// TwinCAT 3 PLC project Untitled1
// ProgramVersion: 3.1.4023.0
// libraries:
//   Tc2_Standard, * (Beckhoff Automation GmbH)
//   Tc2_System, * (Beckhoff Automation GmbH)
//   Tc2_Utilities, * (Beckhoff Automation GmbH)
//   Tc3_Module, * (Beckhoff Automation GmbH)
// project tree:
//   DUTs/ HMI_Instructions.TcDUT, IO_Struct.TcDUT, Port_Map.TcDUT (not stored), Test_Log.TcDUT
//   GVLs/ GVL_HMI.TcGVL, GVL_IO_STRUCTS.TcGVL, GVL_LOGS.TcGVL (not stored), GVL_IO.TcGVL, CONSTANTS.TcGVL
//   / PlcTask.TcTTO (not stored)
//   POUs/ FB_EXECUTE_SECTION1.TcPOU, FB_EXECUTE_SECTION2.TcPOU, INITIALIZE.TcPOU, LOG_SECTION2.TcPOU, LOG_SECTION1.TcPOU, MAIN.TcPOU, UNINITIALIZE.TcPOU, UPDATE_HMI.TcPOU, WRITE_IO_VALUES.TcPOU
// real-time tasks:
//   TASK PlcTask: cycle T#10ms, priority 20, ADS port 350
// I/O:
//   DEVICE Device 1 (EtherCAT), AmsNetId 10.14.22.198.2.1
//     C0 (EK1914) [EK1914, 2 Ch. Safety Input/Output 24V,  TwinSAFE]
//       modules: Module 1 (FSOE), Module 2 (DIO)
//       C1 (EL9410) [EL9410 E-Bus Power Supplier  (Diagnostics)]
//       C2 (EL2014) [EL2014 4Ch. Dig. Output 24V, 0,5A, Diagnostic]
//       C3 (EL1018) [EL1018 8Ch. Dig. Input 24V, 10µs]
//       C4 (EL1819) [EL1819 16Ch. Dig. Input 24V, 10µs]
//       C5 (EL1819) [EL1819 16Ch. Dig. Input 24V, 10µs]
//       C6 (EK1122-0008) [EK1122-0008 2 port EtherCAT junction M8]
//         JBC0 (EK1914) [EK1914, 2 Ch. Safety Input/Output 24V,  TwinSAFE]
//           modules: Module 1 (FSOE), Module 2 (DIO)
//           JBC1 (EL9410) [EL9410 E-Bus Power Supplier  (Diagnostics)]
//           JBC2 (EL1904) [EL1904, 4 Ch. Safety Input 24V, TwinSAFE]
//             modules: Module 1 (FSOES)
//           JBC3 (EL3174) [EL3174 4K. Ana. Eingang  +/-10V Diff., +/-20mA SingleEnded, 16 Bit]
//           JBC4 (EK1122-0008) [EK1122-0008 2 port EtherCAT junction M8]
//           JBC5 (EK1122-0008) [EK1122-0008 2 port EtherCAT junction M8]
//             JBB0 (EP3752-0000) [EP3752-0000 Acceleration Sensor]
// variable links:
//   Untitled1/Untitled1 Instance <-> Device 1 (EtherCAT)/C0 (EK1914)/C2 (EL2014)
//     PlcTask Outputs/GVL_IO.SF5_Fire_Alarm <-> DIG Outputs/Channel 2/Output
//   Untitled1/Untitled1 Instance <-> Device 1 (EtherCAT)/C0 (EK1914)/C3 (EL1018)
//     PlcTask Inputs/GVL_IO.J7_24V_Up <-> Channel 1/Input
//     PlcTask Inputs/GVL_IO.J8_24V_Up <-> Channel 3/Input
//     PlcTask Inputs/GVL_IO.J7_24V_Us <-> Channel 2/Input
//     PlcTask Inputs/GVL_IO.J8_24V_Us <-> Channel 4/Input
//   Untitled1/Untitled1 Instance <-> Device 1 (EtherCAT)/C0 (EK1914)/C4 (EL1819)
//     PlcTask Inputs/GVL_IO.J{1..6}_24V_Up <-> Channel {1..11 step 2}/Input  (6 links)
//     PlcTask Inputs/GVL_IO.J{1..6}_24V_Us <-> Channel {2..12 step 2}/Input  (6 links)
//   Untitled1/Untitled1 Instance <-> Device 1 (EtherCAT)/C0 (EK1914)/C5 (EL1819)
//     PlcTask Inputs/GVL_IO.SF1_MF_CONTINUITY <-> Channel 16/Input
//     PlcTask Inputs/GVL_IO.SF2_MF_CONTINUITY <-> Channel 15/Input
//     PlcTask Inputs/GVL_IO.SF4_Pull_Station <-> Channel 14/Input
//     PlcTask Inputs/GVL_IO.SF6_MGT_CONTINUITY <-> Channel 13/Input
//     PlcTask Inputs/GVL_IO.SF8_MGT_CONTINUITY <-> Channel 12/Input
//   Untitled1/Untitled1 Instance <-> Device 1 (EtherCAT)/C0 (EK1914)/C6 (EK1122-0008)/JBC0 (EK1914)
//     PlcTask Inputs/GVL_IO.JB_DCDCS_OK <-> Module 2 (DIO)/DIO Inputs/Input 0
//     PlcTask Inputs/GVL_IO.JB_Door_Switch <-> Module 2 (DIO)/DIO Inputs/Input 1
//     PlcTask Inputs/GVL_IO.JB_PSU1_OK <-> Module 2 (DIO)/DIO Inputs/Input 2
//     PlcTask Inputs/GVL_IO.JB_PSU2_OK <-> Module 2 (DIO)/DIO Inputs/Input 3

// ---- DUTs/HMI_Instructions.TcDUT
TYPE HMI_Instructions :
STRUCT
	Instructions_Set : STRING(10);
	Instructions : STRING(50);
	Visible : BOOL;
END_STRUCT
END_TYPE

// ---- DUTs/IO_Struct.TcDUT
TYPE IO_Struct :
STRUCT
	SECTION : INT;
	INDEX : INT;
	CARD : STRING(10);
	TERMINAL : USINT;
	SCH_LBL : STRING(10);
	Signal : STRING(25);
	TESTER_PORT : STRING(10);
	TARGET_PORT : STRING(10);
	DESCRIPTION : STRING(255);
	LIVE_BOOL : BOOL;
	LIVE_INT : INT;
	EXPECTED_BOOL : BOOL;
	EXPECTED_INT : INT;
	RESULT : BOOL;
END_STRUCT
END_TYPE

// ---- DUTs/Test_Log.TcDUT
TYPE Test_Log :
STRUCT
	Index : INT;
	Description : STRING(255);
	Result : BOOL;
END_STRUCT
END_TYPE

// ---- GVLs/GVL_HMI.TcGVL
{attribute 'qualified_only'}
VAR_GLOBAL
	
	JBOX_TEST_PORT_MAP : ARRAY[0..CONSTANTS.NUM_CONNECTIONS-1] OF Port_Map := [
		(
			JBOX_PORT := 'J37',
			TESTER_PORT := 'SF1'
		),
		(
			JBOX_PORT := 'S2',
			TESTER_PORT := 'SF2'
		),
		(
			JBOX_PORT := 'S33',
			TESTER_PORT := 'J1'
		),
		(
			JBOX_PORT := 'S34',
			TESTER_PORT := 'J2'
		),
		(
			JBOX_PORT := 'S25',
			TESTER_PORT := 'J3'
		),
		(
			JBOX_PORT := 'S26',
			TESTER_PORT := 'J4'
		),
		(
			JBOX_PORT := 'S27',
			TESTER_PORT := 'J5'
		),
		(
			JBOX_PORT := 'S28',
			TESTER_PORT := 'J6'
		),
		(
			JBOX_PORT := 'S29',
			TESTER_PORT := 'J7'
		),
		(
			JBOX_PORT := 'S30',
			TESTER_PORT := 'J8'
		),
		(
			JBOX_PORT := 'S1',
			TESTER_PORT := 'J9'
		),
		(
			JBOX_PORT := 'S35',
			TESTER_PORT := 'J10'
		),
		(
			JBOX_PORT := 'S3',
			TESTER_PORT := 'J11'
		),
		(
			JBOX_PORT := 'S5',
			TESTER_PORT := 'J12'
		),
		(
			JBOX_PORT := 'S8',
			TESTER_PORT := 'J13'
		),
		(
			JBOX_PORT := 'S10',
			TESTER_PORT := 'J14'
		),
		(
			JBOX_PORT := 'S21',
			TESTER_PORT := 'J15'
		),
		(
			JBOX_PORT := 'S22',
			TESTER_PORT := 'J16'
		),
		(
			JBOX_PORT := 'S23',
			TESTER_PORT := 'J17'
		),
		(
			JBOX_PORT := 'S24',
			TESTER_PORT := 'J18'
		),
		(
			JBOX_PORT := 'S4',
			TESTER_PORT := 'J19'
		),
		(
			JBOX_PORT := 'S6',
			TESTER_PORT := 'J20'
		),
		(
			JBOX_PORT := 'S9',
			TESTER_PORT := 'J21'
		),
		(
			JBOX_PORT := 'S11',
			TESTER_PORT := 'J22'
		),
		(
			JBOX_PORT := 'S13',
			TESTER_PORT := 'J23'
		),
		(
			JBOX_PORT := 'S14',
			TESTER_PORT := 'J24'
		),
		(
			JBOX_PORT := 'S15',
			TESTER_PORT := 'J25'
		),
		(
			JBOX_PORT := 'S16',
			TESTER_PORT := 'J26'
		),
		(
			JBOX_PORT := 'J36',
			TESTER_PORT := 'S17'
		),
		(
			JBOX_PORT := 'J38',
			TESTER_PORT := 'S18'
		)
		];


	
	
	
	
	
	//
	//
	//

	ACTIVE_HMI_VIEW_STRING : STRING(50);
	
	ACTIVE_HMI_VIEW : INT := 0;
	
	HMI_HOME_CONFIRM_CONNECTIONS : BOOL;
	
	HMI_SECTION1_480V_FLASHING : BOOL;
	
	HMI_SECTION1_480V_NOT_FLASHING : BOOL;
	
	HMI_SECTION1_120V_FLASHING : BOOL;
	
	HMI_SECTION1_120V_NOT_FLASHING : BOOL;
	
	HMI_SECTION1_PREP_COMPLETED : BOOL;

	HMI_SECTION1_BEGIN_AUTOMATED : BOOL;
	
	HMI_SECTION2_PREP_COMPLETE : BOOL;
	
	HMI_SECTION2_BEGIN_AUTOMATED : BOOL;
	
	HMI_RESET_JBOX_TEST : BOOL;

	HMI_ABORT_TEST : BOOL;
	
	(*
	HMI_HOME_ACTIVE 			: STRING(10) := 'Hidden';
    HMI_PREP_SECTION1_ACTIVE 	: STRING(10) := 'Hidden';
    HMI_SECTION1_ACTIVE 		: STRING(10) := 'Hidden';
    HMI_PREP_SECTION2_ACTIVE 	: STRING(10) := 'Hidden';
    HMI_SECTION2_ACTIVE 		: STRING(10) := 'Hidden';
    HMI_SECTION999_ACTIVE 		: STRING(10) := 'Hidden';
	*)
	(*
	HMI_HOME_ACTIVE 			: BOOL := FALSE;
    HMI_PREP_SECTION1_ACTIVE 	: BOOL := FALSE;
    HMI_SECTION1_ACTIVE 		: BOOL := FALSE;
    HMI_PREP_SECTION2_ACTIVE 	: BOOL := FALSE;
    HMI_SECTION2_ACTIVE 		: BOOL := FALSE;
    HMI_SECTION999_ACTIVE 		: BOOL := FALSE;
	*)
	


	
	
END_VAR

// ---- GVLs/GVL_IO_STRUCTS.TcGVL
{attribute 'qualified_only'}
VAR_GLOBAL
	
	

	// SECTION ONE OCCURS WITH DOOR CLOSED AND ESTOP DEPRESSED AND NOTHING CONFIGURED
	// NEED TO GET DOOR SWITCH AND ESTOP STUFF IN HERE AT LEAST
	IO_MAP_SECTION1_DIG : ARRAY[0..CONSTANTS.SECTION1_NUM_DIG_TESTS-1] OF IO_STRUCT := [
		(
			SECTION := 1,
			INDEX := 0,
			CARD := 'C3',
			TERMINAL :=  1,
			SCH_LBL := 'SF4',
			SIGNAL := 'Digital',
			TESTER_PORT := 'SF2',
			TARGET_PORT := 'S2',
			DESCRIPTION := 'Fire Pull Station', // This is written to HMI
			LIVE_BOOL := 0, // This is written to from the IO variable
			EXPECTED_BOOL := 1,
			RESULT := 'FAIL' // This is written from HMI
		),
		(
			SECTION := 1,
			INDEX := 1,
			CARD := 'C3',
			TERMINAL :=  2,
			SCH_LBL := 'J7_4',
			SIGNAL := 'Digital',
			TESTER_PORT := 'J7',
			TARGET_PORT := '',
			DESCRIPTION := '24V Power Check', // This is written to HMI
			LIVE_BOOL := 0, // This is written to from the IO variable
			EXPECTED_BOOL := 1,
			RESULT := 'FAIL' // This is written from HMI
		),
		(
			SECTION := 1,
			INDEX := 2,
			CARD := 'C3',
			TERMINAL :=  3,
			SCH_LBL := 'J7_5',
			SIGNAL := 'Digital',
			TESTER_PORT := 'J7',
			TARGET_PORT := '',
			DESCRIPTION := '24V Power Check', // This is written to HMI
			LIVE_BOOL := 0, // This is written to from the IO variable
			EXPECTED_BOOL := 1,
			RESULT := 'FAIL' // This is written from HMI
		),
		(
			SECTION := 1,
			INDEX := 3,
			CARD := 'C3',
			TERMINAL :=  4,
			SCH_LBL := 'J3_1',
			SIGNAL := 'Digital',
			TESTER_PORT := 'J3',
			TARGET_PORT := '',
			DESCRIPTION := '24V Power Check', // This is written to HMI
			LIVE_BOOL := 0, // This is written to from the IO variable
			EXPECTED_BOOL := 1,
			RESULT := 'FAIL' // This is written from HMI
		),
		(
			SECTION := 1,
			INDEX := 4,
			CARD := 'C3',
			TERMINAL :=  5,
			SCH_LBL := 'J3_2',
			SIGNAL := 'Digital',
			TESTER_PORT := 'J3',
			TARGET_PORT := '',
			DESCRIPTION := '24V Power Check', // This is written to HMI
			LIVE_BOOL := 0, // This is written to from the IO variable
			EXPECTED_BOOL := 1,
			RESULT := 'FAIL' // This is written from HMI
		),
		(
			SECTION := 1,
			INDEX := 5,
			CARD := 'C3',
			TERMINAL :=  6,
			SCH_LBL := 'J4_1',
			SIGNAL := 'Digital',
			TESTER_PORT := 'J4',
			TARGET_PORT := '',
			DESCRIPTION := '24V Power Check', // This is written to HMI
			LIVE_BOOL := 0, // This is written to from the IO variable
			EXPECTED_BOOL := 1,
			RESULT := 'FAIL' // This is written from HMI
		),
		(
			SECTION := 1,
			INDEX := 6,
			CARD := 'C3',
			TERMINAL :=  7,
			SCH_LBL := 'J4_2',
			SIGNAL := 'Digital',
			TESTER_PORT := 'J4',
			TARGET_PORT := '',
			DESCRIPTION := '24V Power Check', // This is written to HMI
			LIVE_BOOL := 0, // This is written to from the IO variable
			EXPECTED_BOOL := 1,
			RESULT := 'FAIL' // This is written from HMI
		),
		(
			SECTION := 1,
			INDEX := 7,
			CARD := 'C4',
			TERMINAL :=  1,
			SCH_LBL := 'J5_1',
			SIGNAL := 'Digital',
			TESTER_PORT := 'J5',
			TARGET_PORT := '',
			DESCRIPTION := '24V Power Check', // This is written to HMI
			LIVE_BOOL := 0, // This is written to from the IO variable
			EXPECTED_BOOL := 1,
			RESULT := 'FAIL' // This is written from HMI
		),
		(
			SECTION := 1,
			INDEX := 8,
			CARD := 'C4',
			TERMINAL :=  2,
			SCH_LBL := 'J5_2',
			SIGNAL := 'Digital',
			TESTER_PORT := 'J5',
			TARGET_PORT := '',
			DESCRIPTION := '24V Power Check', // This is written to HMI
			LIVE_BOOL := 0, // This is written to from the IO variable
			EXPECTED_BOOL := 1,
			RESULT := 'FAIL' // This is written from HMI
		),
		(
			SECTION := 1,
			INDEX := 9,
			CARD := 'C4',
			TERMINAL :=  3,
			SCH_LBL := 'J6_1',
			SIGNAL := 'Digital',
			TESTER_PORT := 'J6',
			TARGET_PORT := '',
			DESCRIPTION := '24V Power Check', // This is written to HMI
			LIVE_BOOL := 0, // This is written to from the IO variable
			EXPECTED_BOOL := 1,
			RESULT := 'FAIL' // This is written from HMI
		),
		(
			SECTION := 1,
			INDEX := 10,
			CARD := 'C4',
			TERMINAL :=  4,
			SCH_LBL := 'J6_2',
			SIGNAL := 'Digital',
			TESTER_PORT := 'J6',
			TARGET_PORT := '',
			DESCRIPTION := '24V Power Check', // This is written to HMI
			LIVE_BOOL := 0, // This is written to from the IO variable
			EXPECTED_BOOL := 1,
			RESULT := 'FAIL' // This is written from HMI
		),
		(
			SECTION := 1,
			INDEX := 11,
			CARD := 'C4',
			TERMINAL :=  5,
			SCH_LBL := 'J8_4',
			SIGNAL := 'Digital',
			TESTER_PORT := 'J8',
			TARGET_PORT := '',
			DESCRIPTION := '24V Power Check', // This is written to HMI
			LIVE_BOOL := 0, // This is written to from the IO variable
			EXPECTED_BOOL := 1,
			RESULT := 'FAIL' // This is written from HMI
		),
		(
			SECTION := 1,
			INDEX := 12,
			CARD := 'C4',
			TERMINAL :=  6,
			SCH_LBL := 'J8_5',
			SIGNAL := 'Digital',
			TESTER_PORT := 'J8',
			TARGET_PORT := '',
			DESCRIPTION := '24V Power Check', // This is written to HMI
			LIVE_BOOL := 0, // This is written to from the IO variable
			EXPECTED_BOOL := 1,
			RESULT := 'FAIL' // This is written from HMI
		),
		(
			SECTION := 1,
			INDEX := 13,
			CARD := 'C4',
			TERMINAL :=  7,
			SCH_LBL := 'SF2',
			SIGNAL := 'Digital',
			TESTER_PORT := 'SF2',
			TARGET_PORT := 'S2',
			DESCRIPTION := 'Mine Phone Continuity SF2', // This is written to HMI
			LIVE_BOOL := 0, // This is written to from the IO variable
			EXPECTED_BOOL := 1,
			RESULT := 'FAIL' // This is written from HMI
		),
		(
			SECTION := 1,
			INDEX := 14,
			CARD := 'C4',
			TERMINAL :=  8,
			SCH_LBL := 'SF1',
			SIGNAL := 'Digital',
			TESTER_PORT := 'SF2',
			TARGET_PORT := 'S2',
			DESCRIPTION := 'Mine Phone Continuity SF1', // This is written to HMI
			LIVE_BOOL := 0, // This is written to from the IO variable
			EXPECTED_BOOL := 1,
			RESULT := 'FAIL' // This is written from HMI
		),
		(
			SECTION := 1,
			INDEX := 15,
			CARD := 'C5',
			TERMINAL :=  1,
			SCH_LBL := 'SF6',
			SIGNAL := 'Digital',
			TESTER_PORT := 'SF2',
			TARGET_PORT := 'S2',
			DESCRIPTION := 'MGT Continuity SF6', // This is written to HMI
			LIVE_BOOL := 0, // This is written to from the IO variable
			EXPECTED_BOOL := 1,
			RESULT := 'FAIL' // This is written from HMI
		),
		(
			SECTION := 1,
			INDEX := 16,
			CARD := 'C5',
			TERMINAL :=  2,
			SCH_LBL := 'SF8',
			SIGNAL := 'Digital',
			TESTER_PORT := 'SF2',
			TARGET_PORT := 'S2',
			DESCRIPTION := 'MGT Continuity SF8', // This is written to HMI
			LIVE_BOOL := 0, // This is written to from the IO variable
			EXPECTED_BOOL := 1,
			RESULT := 'FAIL' // This is written from HMI
		),
		(
			SECTION := 1,
			INDEX := 17,
			CARD := 'C5',
			TERMINAL :=  3,
			SCH_LBL := 'J1_1',
			SIGNAL := 'Digital',
			TESTER_PORT := 'J1',
			TARGET_PORT := '',
			DESCRIPTION := '24V Lighting Check', // This is written to HMI
			LIVE_BOOL := 0, // This is written to from the IO variable
			EXPECTED_BOOL := 1,
			RESULT := 'FAIL' // This is written from HMI
		),
		(
			SECTION := 1,
			INDEX := 18,
			CARD := 'C5',
			TERMINAL :=  4,
			SCH_LBL := 'J1_2',
			SIGNAL := 'Digital',
			TESTER_PORT := 'J1',
			TARGET_PORT := '',
			DESCRIPTION := '24V Lighting Check', // This is written to HMI
			LIVE_BOOL := 0, // This is written to from the IO variable
			EXPECTED_BOOL := 1,
			RESULT := 'FAIL' // This is written from HMI
		),
		(
			SECTION := 1,
			INDEX := 19,
			CARD := 'C5',
			TERMINAL :=  5,
			SCH_LBL := 'J2_1',
			SIGNAL := 'Digital',
			TESTER_PORT := 'J2',
			TARGET_PORT := '',
			DESCRIPTION := '24V Lighting Check', // This is written to HMI
			LIVE_BOOL := 0, // This is written to from the IO variable
			EXPECTED_BOOL := 1,
			RESULT := 'FAIL' // This is written from HMI
		),
		(
			SECTION := 1,
			INDEX := 20,
			CARD := 'C5',
			TERMINAL :=  6,
			SCH_LBL := 'J2_2',
			SIGNAL := 'Digital',
			TESTER_PORT := 'J2',
			TARGET_PORT := '',
			DESCRIPTION := '24V Lighting Check', // This is written to HMI
			LIVE_BOOL := 0, // This is written to from the IO variable
			EXPECTED_BOOL := 1,
			RESULT := 'FAIL' // This is written from HMI
		)
	];
	
	IO_MAP_SECTION1_HMI : ARRAY[0..CONSTANTS.SECTION1_NUM_HMI_TESTS-1] OF IO_STRUCT := [
		(
			SECTION := 1,
			INDEX := 0,
			CARD := '',
			// TERMINAL := NULL,
			SCH_LBL := '',
			SIGNAL := 'HMI',
			TESTER_PORT := 'J2',
			TARGET_PORT := '',
			DESCRIPTION := 'JBOX 480V Test', // This is written to HMI
			LIVE_BOOL := 0, // This is written to from the IO variable
			EXPECTED_BOOL := 1,
			RESULT := 'FAIL' // This is written from HMI
		),
		(
			SECTION := 1,
			INDEX := 1,
			CARD := '',
			// TERMINAL := NULL,
			SCH_LBL := '',
			SIGNAL := 'HMI',
			TESTER_PORT := '',
			TARGET_PORT := '',
			DESCRIPTION := 'JBOX 120V Test', // This is written to HMI
			LIVE_BOOL := 0, // This is written to from the IO variable
			EXPECTED_BOOL := 1,
			RESULT := 'FAIL' // This is written from HMI
		)
	];
	

	// SECTION TWO OCCURS WITH DOOR OPEN, ESTOP PRESSED, AND PULL STATION PULLED
	// NEED TO GET DOOR SWITCH AND ESTOP STUFF IN HERE
	IO_MAP_SECTION2_DIG : ARRAY[0..CONSTANTS.SECTION2_NUM_DIG_TESTS-1] OF IO_STRUCT := [
		(
			SECTION := 2,
			INDEX := 0,
			CARD := 'C3',
			TERMINAL :=  1,
			SCH_LBL := 'SF4',
			SIGNAL := 'Digital',
			TESTER_PORT := 'SF2',
			TARGET_PORT := 'S2',
			DESCRIPTION := 'Fire Pull Station', // This is written to HMI
			LIVE_BOOL := 0, // This is written to from the IO variable
			EXPECTED_BOOL := 1,
			RESULT := 'FAIL' // This is written from HMI
		)
		];

END_VAR
		
(*
	IO_MAP : ARRAY[0..GVL.NUM_TESTS-1] OF IO_Struct := [
		(
			INDEX := 0,
			CARD := 'C2',
			TERMINAL := 2,
			SCH_LBL := 'SF5',
			SIGNAL := 'Digital',
			TESTER_PORT := 'SF2',
			TARGET_PORT := 'S2',
			DESCRIPTION := 'Fire Alarm Sounds', // This is written to HMI
			LIVE_BOOL := 0, // This is written to from the IO variable
			LIVE_INT := 0, // This is written to from the IO variable
			RESULT := FALSE // This is written from HMI
		),
		(
			INDEX := 1,
			CARD := 'JBC0',
			TERMINAL := ,
			SCH_LBL := ,
			SIGNAL := 'Digital',
			TESTER_PORT := '',
			TARGET_PORT := '',
			DESCRIPTION := 'JBOX EBUS Us Power Good', // This is written to HMI
			LIVE_BOOL := 0, // This is written to from the IO variable
			LIVE_INT := 0, // This is written to from the IO variable
			RESULT := FALSE // This is written from HMI
		),
		(
			INDEX := 2,
			CARD := 'JBC0',
			TERMINAL := ,
			SCH_LBL := ,
			SIGNAL := 'Digital',
			TESTER_PORT := '',
			TARGET_PORT := '',
			DESCRIPTION := 'JBOX EBUS Up Power Good', // This is written to HMI
			LIVE_BOOL := 0, // This is written to from the IO variable
			LIVE_INT := 0, // This is written to from the IO variable
			RESULT := FALSE // This is written from HMI
		),
		(
			INDEX := 24,
			CARD := 'JBC0',
			TERMINAL :=  3,
			SCH_LBL := '',
			SIGNAL := '',
			TESTER_PORT := '',
			TARGET_PORT := '',
			DESCRIPTION := 'PSU1_OK/1.4B', // This is written to HMI
			LIVE_BOOL := 0, // This is written to from the IO variable
			LIVE_INT := 0, // This is written to from the IO variable
			RESULT := FALSE // This is written from HMI
		),
		(
			INDEX := 25,
			CARD := 'JBC0',
			TERMINAL :=  11,
			SCH_LBL := '',
			SIGNAL := '',
			TESTER_PORT := '',
			TARGET_PORT := '',
			DESCRIPTION := 'PSU2_OK/1.4E', // This is written to HMI
			LIVE_BOOL := 0, // This is written to from the IO variable
			LIVE_INT := 0, // This is written to from the IO variable
			RESULT := FALSE // This is written from HMI
		),
		(
			INDEX := 26,
			CARD := 'JBC3',
			TERMINAL :=  13,
			SCH_LBL := '',
			SIGNAL := '',
			TESTER_PORT := '',
			TARGET_PORT := '',
			DESCRIPTION := 'PSU1_IOUT/1.3B', // This is written to HMI
			LIVE_BOOL := 0, // This is written to from the IO variable
			LIVE_INT := 0, // This is written to from the IO variable
			RESULT := FALSE // This is written from HMI
		),
		(
			INDEX := 27,
			CARD := 'JBC3',
			TERMINAL :=  14,
			SCH_LBL := '',
			SIGNAL := '',
			TESTER_PORT := '',
			TARGET_PORT := '',
			DESCRIPTION := 'PSU2_IOUT/1.3E', // This is written to HMI
			LIVE_BOOL := 0, // This is written to from the IO variable
			LIVE_INT := 0, // This is written to from the IO variable
			RESULT := FALSE // This is written from HMI
		)
		];

END_VAR
*)

// ---- GVLs/GVL_IO.TcGVL
{attribute 'qualified_only'}
VAR_GLOBAL
	
	SECTION1_DIG_INPUTS : ARRAY[0..CONSTANTS.SECTION1_NUM_DIG_TESTS-1] OF POINTER TO BOOL;
	
	SECTION2_DIG_INPUTS : ARRAY[0..CONSTANTS.SECTION2_NUM_DIG_TESTS-1] OF POINTER TO BOOL;
	
	

	C2_P2 AT%Q* : BOOL; //3.1 : BOOL; (*INDEX 0 Fire Alarm Sound SF5 (2024 port 2) *)

	JB_1914_Us AT%I* : BOOL; //8.0 : BOOL; (*INDEX 1 JBOX 1914 Up Power *) // mapping is likely wrong
	JB_1914_Up AT%I* : BOOL; //8.1 : BOOL; (*INDEX 2 JBOX 1914 Us Power *) // mapping is likely wrong
	C3_P1 AT%I* : BOOL; //4.0 : BOOL; (*INDEX 3 Fire pull Station SF4 (1008 (1) port 1) *)
	C3_P2 AT%I* : BOOL; //14.1 : BOOL; (*INDEX 4 24V PWR Check J7 (4) (1008 (1) port 2) *)
    C3_P3 AT%I* : BOOL; //4.2 : BOOL; (*INDEX 5 24V PWR Check J7 (5) (1008 (1) port 3) *)
	C3_P4 AT%I* : BOOL; //14.3 : BOOL; (*INDEX 6 24V PWR Check J3 (1) (1008 (1) port 4) *)
	C3_P5 AT%I* : BOOL; //4.4 : BOOL; (*INDEX 7 24V PWR Check J3 (2) (1008 (1) port 5) *)
    C3_P6 AT%I* : BOOL; //4.5 : BOOL; (*INDEX 8 24V PWR Check J4 (1) (1008 (1) port 6) *)
	
    C3_P7 AT%I* : BOOL; //4.7 : BOOL; (*INDEX 9 24V PWR Check J4 (2) (1008 (1) port 7) *)
    C4_P1 AT%I* : BOOL; //5.0 : BOOL; (*INDEX 10 24V PWR Check J5 (1) (1008 (2) port 1) *)
    C4_P2 AT%I* : BOOL; //5.1 : BOOL; (*INDEX 11 24V PWR Check J5 (2) (1008 (2) port 2) *)
    C4_P3 AT%I* : BOOL; //5.2 : BOOL; (*INDEX 12 24V PWR Check J6 (1) (1008 (2) port 3) *)
    C4_P4 AT%I* : BOOL; //5.3 : BOOL; (*INDEX 13 24V PWR Check J6 (2) (1008 (2) port 4) *)
    C4_P5 AT%I* : BOOL; //5.4 : BOOL; (*INDEX 14 24V PWR Check J8 (4) (1008 (2) port 5) *)
    C4_P6 AT%I* : BOOL; //5.5 : BOOL; (*INDEX 15 24V PWR Check J8 (5) (1008 (2) port 6) *)
	
	C4_P7 AT%I* : BOOL; //5.6 : BOOL; (*INDEX 16 Mine Phone Continuity SF2 (1008 (2) port 7) *)
	C4_P8 AT%I* : BOOL; //5.7 : BOOL; (*INDEX 17 Mine Phone Continuity SF1 (1008 (2) port 8) *)
	C5_P1 AT%I* : BOOL; //6.0 : BOOL; (*INDEX 18 MGT Continuity SF6 (1008 (3) port 1) *)
	C5_P2 AT%I* : BOOL; //6.1: BOOL; (*INDEX 19 MGT Continuity SF8 (1008 (3) port 2) *)
	C5_P3 AT%I* : BOOL; //6.2 : BOOL; (*INDEX 20 Lighting 24V Check J1 (1) (1008 (3) port 3) *)
	C5_P4 AT%I* : BOOL; //6.3 : BOOL; (*INDEX 21 Lighting 24V Check J1 (2) (1008 (3) port 4) *)
	C5_P5 AT%I* : BOOL; //6.4 : BOOL; (*INDEX 22 Lighting 24V Check J2 (1) (1008 (3) port 5) *)
	C5_P6 AT%I* : BOOL; //6.5 : BOOL; (*INDEX 23 Lighting 24V Check J2 (2) (1008 (3) port 6) *)
	
	PSU1_Stat AT%I* : BOOL; //8.2 : BOOL; (*INDEX 24 PSU1_OK/1.4B *)
	PSU2_Stat AT%I* : BOOL; //8.3 : BOOL; (*INDEX 25 PSU2_OK/1.4E *)
	
    PSU1_I AT%I* : BOOL; //10.0 : BOOL; (*INDEX 26 PSU1_IOUT/1.3B *)
    PSU2_I AT%I* : BOOL; //10.1 : BOOL; (*INDEX 27 PSU2_IOUT/1.3E *)
	
	// MAYBE BADDD JBC0_P2 AT%I45.0 : BOOL; (* DCDC_OK/1.6C *)
    
	
	
	
	// INCLINOMETERRRRRR
	
	
	(* FIGURE OUT SAFETY STUFF
	
    JBC0_P10 AT%I45.1 : BOOL; (* Door Switch *)
    JBC0_P7 AT%I40.0 : BOOL; (* SAFE_IN1_I *)
    JBC0_P15 AT%I* : BOOL; (* SAFE_IN2_I *)
    JBC0_P6 AT%I* : BOOL; (* SAFE_IN1_O *)
    JBC0_P14 AT%I* : BOOL; (* SAFE_IN2_O *)
    
   
	*)
	
	
	
	(* MAYBE TEST AND DO THIS FOR THE REST OF THE JBOX CARDS
	
	JB_2014_DIAG_1 AT%I61 : BOOL; (* PSU2_IOUT/1.3E *)
	JB_2014_DIAG_2 AT%I61.4 : BOOL; (* PSU2_IOUT/1.3E *)
	JB_2014_DIAG_3 AT%I62 : BOOL; (* PSU2_IOUT/1.3E *)
	JB_2014_DIAG_4 AT%I62.4 : BOOL; (* PSU2_IOUT/1.3E *)
	JB_2014_COM_FAULT AT%I63.0 : BOOL; (* PSU2_IOUT/1.3E *)
	JB_2014_OVERTEMP AT%I63.1 : BOOL; (* PSU2_IOUT/1.3E *)
	JB_2014_UNDERVOLT AT%I63.2 : BOOL; (* PSU2_IOUT/1.3E *)
	JB_2014_MISS_VOLT AT%I63.3 : BOOL; (* PSU2_IOUT/1.3E *)
	*)


END_VAR

// ---- GVLs/CONSTANTS.TcGVL
{attribute 'qualified_only'}
VAR_GLOBAL CONSTANT
	
	TOTAL_NUM_TESTS : INT := 70;
	
	SECTION1_NUM_DIG_TESTS : INT := 21;
	
	SECTION1_NUM_HMI_TESTS : INT := 2;
	
	SECTION2_NUM_DIG_TESTS : INT := 1;
	
	NUM_CONNECTIONS : INT := 30;
	
END_VAR

// ---- POUs/FB_EXECUTE_SECTION1.TcPOU
FUNCTION_BLOCK FB_EXECUTE_SECTION1
VAR_INPUT
	StartTest : BOOL; // Tells this FB to start its checks
END_VAR

VAR_OUTPUT
	Done : BOOL; // Goes True when FB finishes its checks
END_VAR

VAR_IN_OUT
END_VAR

VAR
	i : INT;	
	state : INT; // internal step for the FB's state machine
	AddStep: INT;
END_VAR

IF StartTest THEN
	Done   := FALSE;
    CASE state OF
        0:
			// DIGITAL INPUTS
			FOR i := 0 TO CONSTANTS.SECTION1_NUM_DIG_TESTS - 1 DO
				IF GVL_IO_STRUCTS.IO_MAP_SECTION1_DIG[i].LIVE_BOOL = GVL_IO_STRUCTS.IO_MAP_SECTION1_DIG[i].EXPECTED_BOOL THEN
					GVL_IO_STRUCTS.IO_MAP_SECTION1_DIG[i].RESULT := 'PASS';
				ELSE
					GVL_IO_STRUCTS.IO_MAP_SECTION1_DIG[i].RESULT := 'FAIL';
				END_IF
			END_FOR
			
			FOR i := 0 TO CONSTANTS.SECTION1_NUM_HMI_TESTS -1 DO
				IF GVL_IO_STRUCTS.IO_MAP_SECTION1_HMI[i].LIVE_BOOL = GVL_IO_STRUCTS.IO_MAP_SECTION1_HMI[i].EXPECTED_BOOL THEN
					GVL_IO_STRUCTS.IO_MAP_SECTION1_HMI[i].RESULT := 'PASS';
				ELSE
					GVL_IO_STRUCTS.IO_MAP_SECTION1_HMI[i].RESULT := 'FAIL';
				END_IF
			END_FOR
			
			state := 999;
            
        999:
            // done
			Done := TRUE;
        ;

    END_CASE;
ELSE
    // if StartTest = FALSE, reset
    Done   := FALSE;
    state  := 0;
END_IF

END_FUNCTION_BLOCK

// ---- POUs/FB_EXECUTE_SECTION2.TcPOU
FUNCTION_BLOCK FB_EXECUTE_SECTION2
VAR_INPUT
	StartTest : BOOL; // Tells this FB to start its checks
END_VAR

VAR_OUTPUT
	Done : BOOL; // Goes True when FB finishes its checks
END_VAR

VAR_IN_OUT
END_VAR

VAR
	i : INT;	
	state : INT; // internal step for the FB's state machine
	AddStep: INT;
END_VAR

IF StartTest THEN
	Done   := FALSE;
    CASE state OF
        0:
			// DIGITAL INPUTS
			FOR i := 0 TO CONSTANTS.SECTION2_NUM_DIG_TESTS - 1 DO
				IF GVL_IO_STRUCTS.IO_MAP_SECTION2_DIG[i].LIVE_BOOL = GVL_IO_STRUCTS.IO_MAP_SECTION2_DIG[i].EXPECTED_BOOL THEN
					GVL_IO_STRUCTS.IO_MAP_SECTION2_DIG[i].RESULT := 'PASS';
				ELSE
					GVL_IO_STRUCTS.IO_MAP_SECTION2_DIG[i].RESULT := 'FAIL';
				END_IF
			END_FOR
			
			state := 999;
            
        999:
            // done
			Done := TRUE;
        ;

    END_CASE;
ELSE
    // if StartTest = FALSE, reset
    Done   := FALSE;
    state  := 0;
END_IF

END_FUNCTION_BLOCK

// ---- POUs/INITIALIZE.TcPOU
FUNCTION INITIALIZE : BOOL
VAR_INPUT
END_VAR
VAR
	i : INT;
END_VAR


GVL_LOGS.NUM_TESTS_LOGGED := 0;


GVL_IO.SECTION1_DIG_INPUTS[0] := ADR(GVL_IO.J7_24V_Up);
GVL_IO.SECTION1_DIG_INPUTS[1] := ADR(GVL_IO.J7_24V_Us);
GVL_IO.SECTION1_DIG_INPUTS[2] := ADR(GVL_IO.J8_24V_Up);
GVL_IO.SECTION1_DIG_INPUTS[3] := ADR(GVL_IO.J8_24V_Us);
GVL_IO.SECTION1_DIG_INPUTS[4] := ADR(GVL_IO.J1_24V_Up);
GVL_IO.SECTION1_DIG_INPUTS[5] := ADR(GVL_IO.J1_24V_Us);
GVL_IO.SECTION1_DIG_INPUTS[6] := ADR(GVL_IO.J2_24V_Up);
GVL_IO.SECTION1_DIG_INPUTS[7] := ADR(GVL_IO.J2_24V_Us);
GVL_IO.SECTION1_DIG_INPUTS[8] := ADR(GVL_IO.J3_24V_Up);
GVL_IO.SECTION1_DIG_INPUTS[9] := ADR(GVL_IO.J3_24V_Us);
GVL_IO.SECTION1_DIG_INPUTS[10] := ADR(GVL_IO.J4_24V_Up);
GVL_IO.SECTION1_DIG_INPUTS[11] := ADR(GVL_IO.J4_24V_Us);
GVL_IO.SECTION1_DIG_INPUTS[12] := ADR(GVL_IO.J5_24V_Up);
GVL_IO.SECTION1_DIG_INPUTS[13] := ADR(GVL_IO.J5_24V_Us);
GVL_IO.SECTION1_DIG_INPUTS[14] := ADR(GVL_IO.J6_24V_Up);
GVL_IO.SECTION1_DIG_INPUTS[15] := ADR(GVL_IO.J6_24V_Us);
GVL_IO.SECTION1_DIG_INPUTS[16] := ADR(GVL_IO.SF1_MF_CONTINUITY);
GVL_IO.SECTION1_DIG_INPUTS[17] := ADR(GVL_IO.SF2_MF_CONTINUITY);
GVL_IO.SECTION1_DIG_INPUTS[18] := ADR(GVL_IO.SF4_Pull_Station);
GVL_IO.SECTION1_DIG_INPUTS[19] := ADR(GVL_IO.SF6_MGT_CONTINUITY);
GVL_IO.SECTION1_DIG_INPUTS[20] := ADR(GVL_IO.SF8_MGT_CONTINUITY);
GVL_IO.SECTION1_DIG_INPUTS[21] := ADR(GVL_IO.JB_Door_Switch);
GVL_IO.SECTION1_DIG_INPUTS[22] := ADR(GVL_IO.JB_DCDCS_OK);
GVL_IO.SECTION1_DIG_INPUTS[23] := ADR(GVL_IO.JB_PSU1_OK);


GVL_IO.SECTION2_DIG_INPUTS[0] := ADR(GVL_IO.SF4_Pull_Station);
GVL_IO.SECTION2_DIG_INPUTS[1] := ADR(GVL_IO.JB_Door_Switch);
GVL_IO.SECTION2_DIG_INPUTS[2] := ADR(GVL_IO.JB_PSU2_OK);
GVL_IO.SECTION2_DIG_INPUTS[3] := ADR(GVL_IO.J7_24V_Up);
GVL_IO.SECTION2_DIG_INPUTS[4] := ADR(GVL_IO.J7_24V_Us);
GVL_IO.SECTION2_DIG_INPUTS[5] := ADR(GVL_IO.J8_24V_Up);
GVL_IO.SECTION2_DIG_INPUTS[6] := ADR(GVL_IO.J8_24V_Us);
GVL_IO.SECTION2_DIG_INPUTS[7] := ADR(GVL_IO.J1_24V_Up);
GVL_IO.SECTION2_DIG_INPUTS[8] := ADR(GVL_IO.J1_24V_Us);
GVL_IO.SECTION2_DIG_INPUTS[9] := ADR(GVL_IO.J2_24V_Up);
GVL_IO.SECTION2_DIG_INPUTS[10] := ADR(GVL_IO.J2_24V_Us);
GVL_IO.SECTION2_DIG_INPUTS[11] := ADR(GVL_IO.J3_24V_Up);
GVL_IO.SECTION2_DIG_INPUTS[12] := ADR(GVL_IO.J3_24V_Us);
GVL_IO.SECTION2_DIG_INPUTS[13] := ADR(GVL_IO.J4_24V_Up);
GVL_IO.SECTION2_DIG_INPUTS[14] := ADR(GVL_IO.J4_24V_Us);
GVL_IO.SECTION2_DIG_INPUTS[15] := ADR(GVL_IO.J5_24V_Up);
GVL_IO.SECTION2_DIG_INPUTS[16] := ADR(GVL_IO.J5_24V_Us);
GVL_IO.SECTION2_DIG_INPUTS[17] := ADR(GVL_IO.J6_24V_Up);
GVL_IO.SECTION2_DIG_INPUTS[18] := ADR(GVL_IO.J6_24V_Us);


INITIALIZE := TRUE;

END_FUNCTION

// ---- POUs/LOG_SECTION2.TcPOU
FUNCTION LOG_SECTION2 : BOOL
VAR_INPUT
END_VAR
VAR
	i : INT;
	j : INT;
	start_index : INT;
	end_index : INT;
END_VAR
VAR_OUTPUT
	Done : BOOL;
END_VAR

Done := FALSE;

start_index := GVL_LOGS.NUM_TESTS_LOGGED;
end_index := start_index + CONSTANTS.SECTION2_NUM_DIG_TESTS-1;

// SECTION 2 DIGITAL INPUTS
FOR i := start_index TO end_index DO
	j := i - start_index;
	GVL_LOGS.TEST_RESULTS_ARRAY[i].DESCRIPTION := GVL_IO_STRUCTS.IO_MAP_SECTION2_DIG[j].DESCRIPTION;
	GVL_LOGS.TEST_RESULTS_ARRAY[i].INDEX := i;
	GVL_LOGS.TEST_RESULTS_ARRAY[i].RESULT := GVL_IO_STRUCTS.IO_MAP_SECTION2_DIG[j].RESULT;
	GVL_LOGS.NUM_TESTS_LOGGED := GVL_LOGS.NUM_TESTS_LOGGED + 1;
END_FOR

Done := TRUE;

END_FUNCTION

// ---- POUs/LOG_SECTION1.TcPOU
FUNCTION LOG_SECTION1 : BOOL
VAR_INPUT
END_VAR
VAR
	i : INT;
	j : INT;
	start_index : INT;
	end_index : INT;
END_VAR

start_index := GVL_LOGS.NUM_TESTS_LOGGED;
end_index := start_index + CONSTANTS.SECTION1_NUM_DIG_TESTS-1;

// SECTION 3 DIGITAL INPUTS
FOR i := start_index TO end_index DO
	j := i - start_index;
	GVL_LOGS.TEST_RESULTS_ARRAY[i].DESCRIPTION := GVL_IO_STRUCTS.IO_MAP_SECTION1_DIG[j].DESCRIPTION;
	GVL_LOGS.TEST_RESULTS_ARRAY[i].INDEX := i;
	GVL_LOGS.TEST_RESULTS_ARRAY[i].RESULT := GVL_IO_STRUCTS.IO_MAP_SECTION1_DIG[j].RESULT;
	GVL_LOGS.NUM_TESTS_LOGGED := GVL_LOGS.NUM_TESTS_LOGGED + 1;
END_FOR

END_FUNCTION

// ---- POUs/MAIN.TcPOU
PROGRAM MAIN
VAR_INPUT
END_VAR
VAR
	ExecuteSection1 : FB_EXECUTE_SECTION1;
	ExecuteSection2 : FB_EXECUTE_SECTION2;

END_VAR


IF GVL_HMI.HMI_ABORT_TEST THEN
	UNINITIALIZE();
END_IF

CASE GVL_HMI.ACTIVE_HMI_VIEW OF
  0: GVL_HMI.ACTIVE_HMI_VIEW_STRING := 'Home_Page.content';
  1: GVL_HMI.ACTIVE_HMI_VIEW_STRING := 'Section_1.content';
  2: GVL_HMI.ACTIVE_HMI_VIEW_STRING := 'Section_2.content';
  3: GVL_HMI.ACTIVE_HMI_VIEW_STRING := 'Results_Page.content';
  ELSE GVL_HMI.ACTIVE_HMI_VIEW_STRING := 'Home_Page.content';  // default
END_CASE;

CASE GVL_HMI.ACTIVE_HMI_VIEW OF
	
	0: // Idle
	
		Initialize();
		Update_HMI();
		
		IF GVL_HMI.HMI_HOME_CONFIRM_CONNECTIONS THEN
			GVL_HMI.ACTIVE_HMI_VIEW := 1;
			Update_HMI();
		END_IF
		
	1: 
		IF GVL_HMI.HMI_SECTION1_PREP_COMPLETED THEN
			GVL_HMI.ACTIVE_HMI_VIEW := 2;
			Update_HMI();
		END_IF
		
	2:
		
		IF GVL_HMI.HMI_SECTION1_BEGIN_AUTOMATED THEN
			WRITE_IO_VALUES();
			ExecuteSection1(StartTest := TRUE);
			IF ExecuteSection1.Done THEN
				LOG_SECTION1();

				Update_HMI();
				GVL_HMI.ACTIVE_HMI_VIEW := 3;

			END_IF

		END_IF
		
	3:
		IF GVL_HMI.HMI_SECTION2_PREP_COMPLETE THEN
			GVL_HMI.ACTIVE_HMI_VIEW := 4;
			Update_HMI();
		END_IF
		
	4: 
		IF GVL_HMI.HMI_SECTION2_BEGIN_AUTOMATED THEN
			IF WRITE_IO_VALUES() THEN
				ExecuteSection2(StartTest := TRUE);
				IF ExecuteSection2.Done THEN
					LOG_SECTION2();

					Update_HMI();
					GVL_HMI.ACTIVE_HMI_VIEW := 5;
				END_IF
			END_IF
		END_IF
		
	5: // Test done
		IF GVL_HMI.HMI_RESET_JBOX_TEST THEN
			UNINITIALIZE();
		END_IF

		
		
END_CASE

END_PROGRAM

// ---- POUs/UNINITIALIZE.TcPOU
FUNCTION UNINITIALIZE : BOOL
VAR_INPUT
END_VAR
VAR
	i : INT;
END_VAR



	
FOR i := 0 TO CONSTANTS.SECTION1_NUM_DIG_TESTS - 1 DO
	GVL_IO_STRUCTS.IO_MAP_SECTION1_DIG[i].LIVE_BOOL := FALSE;
	GVL_IO_STRUCTS.IO_MAP_SECTION1_DIG[i].Result := 'FAIL';
END_FOR

FOR i := 0 TO CONSTANTS.SECTION1_NUM_HMI_TESTS - 1 DO
	GVL_IO_STRUCTS.IO_MAP_SECTION1_HMI[i].LIVE_BOOL := FALSE;
	GVL_IO_STRUCTS.IO_MAP_SECTION1_HMI[i].Result := 'FAIL';
END_FOR

FOR i := 0 TO CONSTANTS.SECTION2_NUM_DIG_TESTS - 1 DO
	GVL_IO_STRUCTS.IO_MAP_SECTION2_DIG[i].LIVE_BOOL := FALSE;
	GVL_IO_STRUCTS.IO_MAP_SECTION2_DIG[i].Result := 'FAIL';
END_FOR


FOR I := 0 TO GVL_LOGS.NUM_TESTS_LOGGED - 1 DO
	GVL_LOGS.TEST_RESULTS_ARRAY[i].Description := '';
	GVL_LOGS.TEST_RESULTS_ARRAY[i].Index := 0;
	GVL_LOGS.TEST_RESULTS_ARRAY[i].Result := '';
END_FOR

GVL_LOGS.NUM_TESTS_LOGGED := 0;

GVL_HMI.ACTIVE_HMI_VIEW := 0;
UPDATE_HMI();


Uninitialize := TRUE;

END_FUNCTION

// ---- POUs/UPDATE_HMI.TcPOU
FUNCTION UPDATE_HMI : BOOL
VAR_INPUT
END_VAR
VAR
END_VAR


(*
CASE GVL_HMI.ACTIVE_HMI_VIEW OF
	
	0:
		GVL_HMI.HMI_HOME_ACTIVE 			:= TRUE;
    	GVL_HMI.HMI_PREP_SECTION1_ACTIVE 	:= FALSE;
    	GVL_HMI.HMI_SECTION1_ACTIVE 		:= FALSE;
    	GVL_HMI.HMI_PREP_SECTION2_ACTIVE 	:= FALSE;
    	GVL_HMI.HMI_SECTION2_ACTIVE 		:= FALSE;
   		GVL_HMI.HMI_SECTION999_ACTIVE 		:= FALSE;
	1:
		GVL_HMI.HMI_HOME_ACTIVE 			:= FALSE;
    	GVL_HMI.HMI_PREP_SECTION1_ACTIVE 	:= TRUE;
    	GVL_HMI.HMI_SECTION1_ACTIVE 		:= FALSE;
    	GVL_HMI.HMI_PREP_SECTION2_ACTIVE 	:= FALSE;
    	GVL_HMI.HMI_SECTION2_ACTIVE 		:= FALSE;
   		GVL_HMI.HMI_SECTION999_ACTIVE 		:= FALSE;
	2:
		GVL_HMI.HMI_HOME_ACTIVE 			:= FALSE;
    	GVL_HMI.HMI_PREP_SECTION1_ACTIVE 	:= FALSE;
    	GVL_HMI.HMI_SECTION1_ACTIVE 		:= TRUE;
    	GVL_HMI.HMI_PREP_SECTION2_ACTIVE 	:= FALSE;
    	GVL_HMI.HMI_SECTION2_ACTIVE 		:= FALSE;
   		GVL_HMI.HMI_SECTION999_ACTIVE 		:= FALSE;
	3:
		GVL_HMI.HMI_HOME_ACTIVE 			:= FALSE;
    	GVL_HMI.HMI_PREP_SECTION1_ACTIVE 	:= FALSE;
    	GVL_HMI.HMI_SECTION1_ACTIVE 		:= FALSE;
    	GVL_HMI.HMI_PREP_SECTION2_ACTIVE 	:= TRUE;
    	GVL_HMI.HMI_SECTION2_ACTIVE 		:= FALSE;
   		GVL_HMI.HMI_SECTION999_ACTIVE 		:= FALSE;
	4:
		GVL_HMI.HMI_HOME_ACTIVE 			:= FALSE;
    	GVL_HMI.HMI_PREP_SECTION1_ACTIVE 	:= FALSE;
    	GVL_HMI.HMI_SECTION1_ACTIVE 		:= FALSE;
    	GVL_HMI.HMI_PREP_SECTION2_ACTIVE 	:= FALSE;
    	GVL_HMI.HMI_SECTION2_ACTIVE 		:= TRUE;
   		GVL_HMI.HMI_SECTION999_ACTIVE 		:= FALSE;
	5:
		GVL_HMI.HMI_HOME_ACTIVE 			:= FALSE;
    	GVL_HMI.HMI_PREP_SECTION1_ACTIVE 	:= FALSE;
    	GVL_HMI.HMI_SECTION1_ACTIVE 		:= FALSE;
    	GVL_HMI.HMI_PREP_SECTION2_ACTIVE 	:= FALSE;
    	GVL_HMI.HMI_SECTION2_ACTIVE 		:= FALSE;
   		GVL_HMI.HMI_SECTION999_ACTIVE 		:= TRUE;
	
END_CASE
*)

END_FUNCTION

// ---- POUs/WRITE_IO_VALUES.TcPOU
FUNCTION WRITE_IO_VALUES : BOOL
VAR_INPUT
END_VAR
VAR
	i : INT;
END_VAR


// Write Values to IO Structures

// WRITE VALUES TO SECTION 1 Digital Input VARIABLES
FOR i := 0 TO CONSTANTS.SECTION1_NUM_DIG_TESTS - 1 DO
	GVL_IO_STRUCTS.IO_MAP_SECTION1_DIG[i].LIVE_BOOL := GVL_IO.SECTION1_DIG_INPUTS[i]^;
END_FOR



// WRITE VALUES TO SECTION 2 Digital Input Variables
FOR i := 0 TO CONSTANTS.SECTION2_NUM_DIG_TESTS - 1 DO
	GVL_IO_STRUCTS.IO_MAP_SECTION2_DIG[i].LIVE_BOOL := GVL_IO.SECTION2_DIG_INPUTS[i]^;
END_FOR



WRITE_IO_VALUES := TRUE;


// Write Values to other test variables


(*
GVL_IO_STRUCTS.FIRE_ALRM_P5.LIVE_BOOL := GVL_IO.C2_P2;
GVL_IO_STRUCTS.JB_CARD_Us.LIVE_BOOL := GVL_IO.JB_1914_Us;
GVL_IO_STRUCTS.JB_CARD_Up.LIVE_BOOL := GVL_IO.JB_1914_Up;
GVL_IO_STRUCTS.FIRE_PULL_P4.LIVE_BOOL := GVL_IO.C3_P1;
GVL_IO_STRUCTS.Us_24V_5.LIVE_BOOL := GVL_IO.C3_P2;
GVL_IO_STRUCTS.Up_24V_5.LIVE_BOOL := GVL_IO.C3_P3;
GVL_IO_STRUCTS.Us_24V_1.LIVE_BOOL := GVL_IO.C3_P4;
GVL_IO_STRUCTS.Up_24V_1.LIVE_BOOL := GVL_IO.C3_P5;
GVL_IO_STRUCTS.Us_24V_2.LIVE_BOOL := GVL_IO.C3_P6;
GVL_IO_STRUCTS.Up_24V_2.LIVE_BOOL := GVL_IO.C3_P7;
GVL_IO_STRUCTS.Us_24V_3.LIVE_BOOL := GVL_IO.C4_P1;
GVL_IO_STRUCTS.Up_24V_3.LIVE_BOOL := GVL_IO.C4_P2;
GVL_IO_STRUCTS.Us_24V_4.LIVE_BOOL := GVL_IO.C4_P3;
GVL_IO_STRUCTS.Up_24V_4.LIVE_BOOL := GVL_IO.C4_P4;
GVL_IO_STRUCTS.Us_24V_6.LIVE_BOOL := GVL_IO.C4_P5;
GVL_IO_STRUCTS.Up_24V_6.LIVE_BOOL := GVL_IO.C4_P6;
GVL_IO_STRUCTS.PHONE_P2.LIVE_BOOL := GVL_IO.C4_P7;
GVL_IO_STRUCTS.PHONE_P1.LIVE_BOOL := GVL_IO.C4_P8;
GVL_IO_STRUCTS.MGT_P6.LIVE_BOOL := GVL_IO.C5_P1;
GVL_IO_STRUCTS.MGT_P8.LIVE_BOOL := GVL_IO.C5_P2;
GVL_IO_STRUCTS.LIGHT_24V_Us_1.LIVE_BOOL := GVL_IO.C5_P3;
GVL_IO_STRUCTS.LIGHT_24V_Up_1.LIVE_BOOL := GVL_IO.C5_P4;
GVL_IO_STRUCTS.LIGHT_24V_Us_2.LIVE_BOOL := GVL_IO.C5_P5;
GVL_IO_STRUCTS.LIGHT_24V_Up_2.LIVE_BOOL := GVL_IO.C5_P6;
*)

END_FUNCTION
